// TIA Portal V16 export
// export: Created 2023-03-29T11:03:44.988455Z, ExportSetting WithDefaults, DisplayName Totally Integrated Automation Portal, DisplayVersion V16 Update 6, DisplayName TIA Portal Version Control Interface, DisplayVersion V16 Update 2, DisplayName TIA Portal Openness, DisplayVersion V16 Update 6, DisplayName STEP 7 Professional, DisplayVersion V16 Update 6, DisplayName STEP 7 Safety, DisplayVersion V16, DisplayName WinCC Advanced, DisplayVersion V16 Update 6
VAR_GLOBAL   // PLC tag table "Z5"
   inputAwariaMomentZ_5 AT %M62.5 : Bool;   // znacznik wejście
   inputRuch_Z_5 AT %M62.4 : Bool;
   inputAumalokalneZ_5 AT %M62.6 : Bool;   // znacznik wejście
   Hbit_Zamknij_Z5 AT %M18.5 : Bool;
   inputOtwartaZ_5 AT %M62.2 : Bool;   // znacznik wejście
   Hbit_Otwarta_Z5 AT %M18.1 : Bool;
   setSVMC_Z_5 AT %M63.3 : Bool;   // Znacznik polecenia zamknij w trybie automat
   CMD_Close_Z_5 AT %M63.6 : Bool;   // załącz zamykanie
   inputAumaautomatZ_5 AT %M62.7 : Bool;   // znacznik wejście
   Hbit_Auto_Manu_Z5 AT %M18.7 : Bool;
   CMD_Open_Z_5 AT %M63.5 : Bool;   // załącz otwieranie
   inputAumagotowośćZ_5 AT %M63.0 : Bool;   // znacznik wejście
   CMD_Awaria_Z_5 AT %M63.7 : Bool;   // Awaria zbiorcza
   setSVMO_Z_5 AT %M63.2 : Bool;   // Znacznik polecenia otwórz w trybie automat
   Hbit_Zamknieta_Z5 AT %M18.3 : Bool;
   Hbit_Alarm_Z5 AT %M18.0 : Bool;
   isAUMA_Z_5 AT %M52.6 : Bool;   // przęłącznik wymiany na AUMA
   inputAumaawariaZ_5 AT %M63.1 : Bool;   // znacznik wejście
   Hbit_Reset_Z5 AT %M18.6 : Bool;
   isGotowość_Z_5 AT %M62.0 : Bool;   // bit gotowości wspólny
   Byte_Status_Z5 AT %MW18 : Word;   // Słowo statusu napędu
   Hbit_REN_Z5 AT %M18.2 : Bool;
   inputREMT_Z_5 AT %M62.1 : Bool;   // znacznik wejście zdalne
   inputZamkniętaZ_5 AT %M62.3 : Bool;   // znacznik wejście
   setAlarm_Moment_Z_5 AT %M63.4 : Bool;   // znacznik alarmu od momentówki w trybie zdalnym (aut/mamnual)
   Hbit_Otwórz_Z5 AT %M18.4 : Bool;
END_VAR
